Staubli VAL3: S2S_demo_1.pjx

--- S2S_demo_1.pjx ---
Parameters version=s7.9.1 stackSize=5000 millimeterUnit=true
Program file=start.pgx
Program file=stop.pgx
Program file=updateCycleNum.pgx
Program file=waitPLCstart.pgx
Data file=S2S_demo_1.dtx
Library alias=S7 path=Disk://S2S/S2S.pjx autoload=true password=

--- S2S_demo_1.dtx ---
mdesc mNomSpeed
num nDB[100]
  [0] = 1
  [1] = 2
  [2] = 3
  [3] = 4
  [4] = 5
  [5] = 6
  [6] = 7
  [7] = 8
  [8] = 9
  [9] = 10
  [10] = 1
  [11] = 2
  [12] = 3
  [13] = 4
  [14] = 5
  [15] = 6
  [16] = 7
  [17] = 8
  [18] = 9
  [19] = 10
  [20] = 1
  [21] = 2
  [22] = 3
  [23] = 4
  [24] = 5
  [25] = 6
  [26] = 7
  [27] = 8
  [28] = 9
  [29] = 10
  [30] = 1
  [31] = 2
  [32] = 3
  [33] = 4
  [34] = 5
  [35] = 6
  [36] = 7
  [37] = 8
  [38] = 9
  [39] = 10
  [40] = 1
  [41] = 2
  [42] = 3
  [43] = 4
  [44] = 5
  [45] = 6
  [46] = 7
  [47] = 8
  [48] = 9
  [49] = 10
  [50] = 1
  [51] = 2
  [52] = 3
  [53] = 4
  [54] = 5
  [55] = 6
  [56] = 7
  [57] = 8
  [58] = 9
  [59] = 10
  [60] = 1
  [61] = 2
  [62] = 3
  [63] = 4
  [64] = 5
  [65] = 6
  [66] = 7
  [67] = 8
  [68] = 9
  [69] = 10
  [70] = 1
  [71] = 2
  [72] = 3
  [73] = 4
  [74] = 5
  [75] = 6
  [76] = 7
  [77] = 8
  [78] = 9
  [79] = 10
  [80] = 1
  [81] = 2
  [82] = 3
  [83] = 4
  [84] = 5
  [85] = 6
  [86] = 7
  [87] = 8
  [88] = 9
  [89] = 10
  [90] = 1
  [91] = 2
  [92] = 3
  [93] = 4
  [94] = 5
  [95] = 6
  [96] = 7
  [97] = 8
  [98] = 9
  [99] = 10
num nDBread = 1
num nDBwrite = 2
pointRx pPick = {x=-279.850434, y=86.377812, z=-61.0164915, rx=0.00168696, ry=179.999787, rz=-87.79852, shoulder=righty, elbow=enegative, wrist=wpositive, fatherId=world[0]}
pointRx pPlace = {x=-223.225508, y=308.777671, z=-61.0164596, rx=0.00255065, ry=-179.999305, rz=-87.798275, shoulder=righty, elbow=enegative, wrist=wpositive, fatherId=world[0]}
sio sTcpClient = {link=Socket\sTcpClient}

--- start.pgx ---
program start()
  local num l_nCycleNum
begin

  //the purpose of this demo is to give a minimal example of a good "workflow" for the use of this library
  //For this example we must have two separated db's on plc side: one to read data from plc and the other to write data to plc

  cls()
  call S7:init(sTcpClient)
  call S7:connectTo("127.0.0.1",0,2)

  l_nCycleNum=0
  if S7:nLastError==S7:nNoErrors
    while true

      call waitPLCstart()
      movej(appro(pPick,{0,0,-50,0,0,0}),flange,mNomSpeed)
      movel(pPick,flange,mNomSpeed)
      movel(appro(pPick,{0,0,-50,0,0,0}),flange,mNomSpeed)
      movej(appro(pPlace,{0,0,-50,0,0,0}),flange,mNomSpeed)
      movel(pPlace,flange,mNomSpeed)
      movel(appro(pPlace,{0,0,-50,0,0,0}),flange,mNomSpeed)
      waitEndMove()
      l_nCycleNum=l_nCycleNum+1
      call updateCycleNum(l_nCycleNum)
    endWhile
  else
    userPage()
    putln("error during connection")
  endIf

end

--- stop.pgx ---
program stop()
begin
end

--- updateCycleNum.pgx ---
program updateCycleNum(num x_nNum (dimensions=1))
  local num l_nLocalWord[2]
begin

  //let's suppose that in the plc's db "nDBwrite" there is a word, starting from byte 10, that represent the number of cyle performed by
  //the robot

  //first of all we have to "translate" the argument x_nNum in a 2 byte buffer representing the word (using "big-endian" format)
  //the better way to do this is a local 2 elements array written by the "helper" function setWordAt
  call S7:setWordAt(0,x_nNum,l_nLocalWord)

  //then we write this buffer to nDBwrite!
  call S7:writeArea(S7:nAreaDB,nDBwrite,l_nLocalWord,0,size(l_nLocalWord))

end

--- waitPLCstart.pgx ---
program waitPLCstart()
  local bool l_bRes
  local num l_nRes
begin

  //let's suppose the "start bit" is in the third byte, 5th bit of "nDBread" on plc-side
  //
  //  nDBread:
  //    byte0:  bit0 bit1 bit2 bit3 bit4 bit5 bit6 bit7
  //    byte1:  bit0 bit1 bit2 bit3 bit4 bit5 bit6 bit7
  //    byte2:  bit0 bit1 bit2 bit3 "bStartRobot" bit5 bit6 bit7

  l_bRes=false
  do
    //i just need to read starting from the 3th byte (counting from 0) one byte from "nDBread" and put it into l_nRes
    call S7:readArea(S7:nAreaDB,nDBread,2,1,l_nRes)
    //now i get the 5th bit (counting from 0) value from the beginning (0) of the "buffer" l_nRes
    call S7:getBitAt(0,4,l_nRes,l_bRes)
    delay(0)
  until l_bRes


end
